FUNCTION_BLOCK Analysis
VAR
	arnNumberArray : ARRAY[0..7] OF UINT;
END_VAR

METHOD AnalyzeLine
VAR_INPUT
	sTextLine : STRING;
END_VAR
VAR_OUTPUT
	bIncreasing : BOOL;
	bDecreasing : BOOL;
	bClose : BOOL;
END_VAR
VAR
	sCurrentString : STRING;
	sSubString : STRING;
	nIndexOfNextSpace : INT;
	nLoopIndex : UINT;
END_VAR
sSubString := sTextLine;
nIndexOfNextSpace := FIND(sSubString, ' ');
nLoopIndex := 0;
WHILE nIndexOfNextSpace > 0 DO
	sCurrentString := LEFT(sSubString, nIndexOfNextSpace-1);
	sSubString := RIGHT(sSubString, LEN(sSubString)-nIndexOfNextSpace);
	arnNumberArray[nLoopIndex] := TO_UINT(sCurrentString);
	nIndexOfNextSpace:= FIND(sSubString, ' ');
	nLoopIndex := nLoopIndex;
END_WHILE
arnNumberArray[nLoopIndex+1] := TO_UINT(sSubString);
bIncreasing := THIS^.CheckIncreasing(nLoopIndex+1);
bDecreasing := THIS^.CheckDecreasing(nLoopIndex+1);
bClose := THIS^.CheckClose(nLoopIndex+1);
END_METHOD

METHOD CheckClose : BOOL
VAR_INPUT
	nNumElementsInLine : UINT;
END_VAR
VAR
	iLoopIndex : UINT;
	nDistance : INT;
	bStepClose : BOOL;
	bAllClose : BOOL;
END_VAR
bAllClose := TRUE;
FOR iLoopIndex := 0 TO nNumElementsInLine-2 DO
	nDistance := arnNumberArray[iLoopIndex] - arnNumberArray[iLoopIndex+1];
	nDistance := ABS(nDistance);
	bStepClose := nDistance >= 1 AND nDistance <=3; 
	bAllClose := bAllClose AND bStepClose;			
END_FOR
CheckClose := bAllClose;
END_METHOD

METHOD CheckDecreasing : BOOL
VAR_INPUT
	nNumElementsInLine : UINT;
END_VAR
VAR
	iLoopIndex : UINT;
	bStepDecreasing : BOOL;
	bStrictlyDecreasing : BOOL;
END_VAR
bStrictlyDecreasing := TRUE;
FOR iLoopIndex := 0 TO nNumElementsInLine-2 DO
	bStepDecreasing := arnNumberArray[iLoopIndex] > arnNumberArray[iLoopIndex+1];
	bStrictlyDecreasing := bStrictlyDecreasing AND bStepDecreasing;			
END_FOR
CheckDecreasing := bStrictlyDecreasing;
END_METHOD

METHOD CheckIncreasing : BOOL
VAR_INPUT
	nNumElementsInLine : UINT;
END_VAR
VAR
	iLoopIndex : UINT;
	bStepIncreasing : BOOL;
	bStrictlyIncreasing : BOOL;
END_VAR
bStrictlyIncreasing := TRUE;
FOR iLoopIndex := 0 TO nNumElementsInLine-2 DO
	bStepIncreasing := arnNumberArray[iLoopIndex] < arnNumberArray[iLoopIndex+1];
	bStrictlyIncreasing := bStrictlyIncreasing AND bStepIncreasing;			
END_FOR
CheckIncreasing := bStrictlyIncreasing;
END_METHOD

END_FUNCTION_BLOCK

(* stored: Version 1.1.0.1
   POU Analysis: Id {1d1e40ed-f79c-44df-ac24-3b472246fdc9}, SpecialFunc None
   Method AnalyzeLine: Id {b8d78072-f55e-417c-9fa4-5dcbaada27eb}
   Method CheckClose: Id {f6c18ddd-5609-419d-b098-cf14392fc482}
   Method CheckDecreasing: Id {31cdb210-42b1-49f8-906a-93cd577c0ab4}
   Method CheckIncreasing: Id {1bb71b02-f0ac-4030-946c-d08e773724bd} *)
